{attribute 'GeneratedUsingTerminal: KL6224'}
{attribute addProperty BoxType "KL6224"}
{attribute addProperty Id "StatusAT %I*UINT0Parameter_InAT %I*UDINT0State_Ch1AT %I*USINT0State_Ch2AT %I*USINT0State_Ch3AT %I*USINT0State_Ch4AT %I*USINT0Data_In_0AT %I*USINT0Data_In_1AT %I*USINT0ControlAT %Q*UINT0Parameter_OutAT %Q*UDINT0Data_Out_0AT %Q*USINT0Data_Out_1AT %Q*USINT0Data_Out_2AT %Q*USINT0Data_Out_3AT %Q*USINT0Data_Out_4AT %Q*USINT0Data_Out_5AT %Q*USINT0"}
{attribute addProperty CRC "139488206"}
{attribute addProperty Size "0"}
TYPE Channel_08506BCE :
STRUCT
	{attribute addProperty Name "Status"}
	Status AT %I* : UINT;
	{attribute addProperty Name "Parameter_In"}
	Parameter_In AT %I* : UDINT;
	{attribute addProperty Name "State_Ch1"}
	State_Ch1 AT %I* : USINT;
	{attribute addProperty Name "State_Ch2"}
	State_Ch2 AT %I* : USINT;
	{attribute addProperty Name "State_Ch3"}
	State_Ch3 AT %I* : USINT;
	{attribute addProperty Name "State_Ch4"}
	State_Ch4 AT %I* : USINT;
	{attribute addProperty Name "Data_In_0"}
	Data_In_0 AT %I* : USINT;
	{attribute addProperty Name "Data_In_1"}
	Data_In_1 AT %I* : USINT;
	{attribute addProperty Name "Control"}
	Control AT %Q* : UINT;
	{attribute addProperty Name "Parameter_Out"}
	Parameter_Out AT %Q* : UDINT;
	{attribute addProperty Name "Data_Out_0"}
	Data_Out_0 AT %Q* : USINT;
	{attribute addProperty Name "Data_Out_1"}
	Data_Out_1 AT %Q* : USINT;
	{attribute addProperty Name "Data_Out_2"}
	Data_Out_2 AT %Q* : USINT;
	{attribute addProperty Name "Data_Out_3"}
	Data_Out_3 AT %Q* : USINT;
	{attribute addProperty Name "Data_Out_4"}
	Data_Out_4 AT %Q* : USINT;
	{attribute addProperty Name "Data_Out_5"}
	Data_Out_5 AT %Q* : USINT;
END_STRUCT
END_TYPE

(* stored: Version 1.2.0.0, ProductVersion 3.1.4024.9
   DUT Channel_08506BCE: Id {7400396a-b28a-4a76-9bd6-052fc7ff0969} *)
